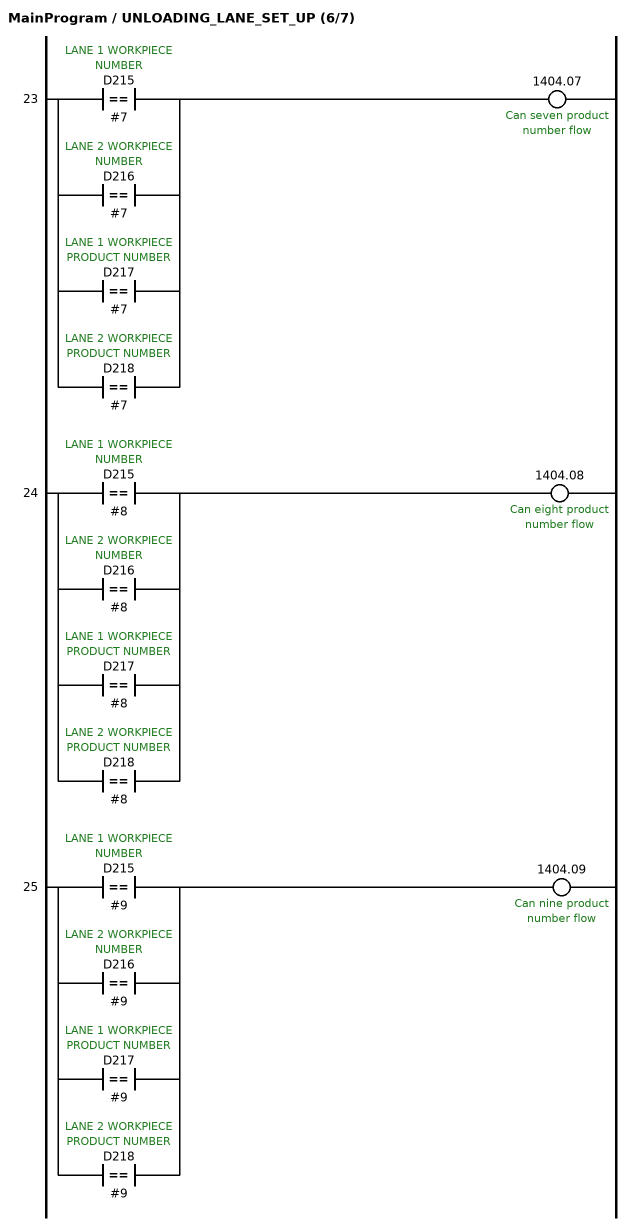
; [picture p192: MainProgram / UNLOADING_LANE_SET_UP, rungs 23-25]
; rung 23
LD=(300) D215 #7  ; LANE 1 WORKPIECE NUMBER
OR=(300) D216 #7  ; LANE 2 WORKPIECE NUMBER
OR=(300) D217 #7  ; LANE 1 WORKPIECE PRODUCT NUMBER
OR=(300) D218 #7  ; LANE 2 WORKPIECE PRODUCT NUMBER
OUT 1404.07  ; Can seven product number flow
; rung 24
LD=(300) D215 #8  ; LANE 1 WORKPIECE NUMBER
OR=(300) D216 #8  ; LANE 2 WORKPIECE NUMBER
OR=(300) D217 #8  ; LANE 1 WORKPIECE PRODUCT NUMBER
OR=(300) D218 #8  ; LANE 2 WORKPIECE PRODUCT NUMBER
OUT 1404.08  ; Can eight product number flow
; rung 25
LD=(300) D215 #9  ; LANE 1 WORKPIECE NUMBER
OR=(300) D216 #9  ; LANE 2 WORKPIECE NUMBER
OR=(300) D217 #9  ; LANE 1 WORKPIECE PRODUCT NUMBER
OR=(300) D218 #9  ; LANE 2 WORKPIECE PRODUCT NUMBER
OUT 1404.09  ; Can nine product number flow

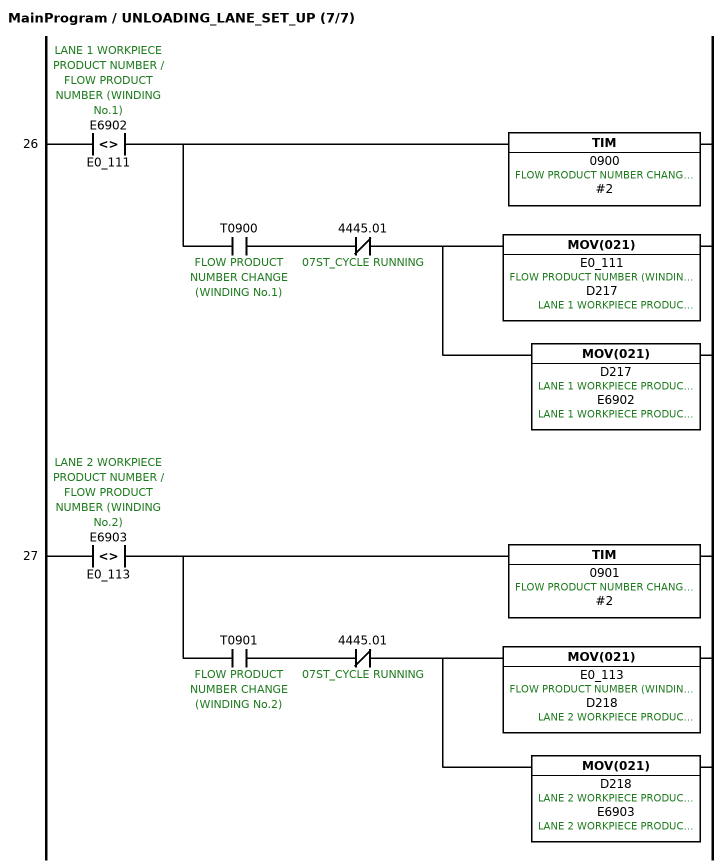
; rung 26
LD<>(305) E6902 E0_111  ; LANE 1 WORKPIECE PRODUCT NUMBER, FLOW PRODUCT NUMBER (WINDING No.1)
TIM 0900 #2  ; FLOW PRODUCT NUMBER CHANGE (WINDING No.1)
AND T0900  ; FLOW PRODUCT NUMBER CHANGE (WINDING No.1)
ANDNOT 4445.01  ; 07ST_CYCLE RUNNING
MOV(021) E0_111 D217  ; FLOW PRODUCT NUMBER (WINDING No.1), LANE 1 WORKPIECE PRODUCT NUMBER
MOV(021) D217 E6902  ; LANE 1 WORKPIECE PRODUCT NUMBER
; rung 27
LD<>(305) E6903 E0_113  ; LANE 2 WORKPIECE PRODUCT NUMBER, FLOW PRODUCT NUMBER (WINDING No.2)
TIM 0901 #2  ; FLOW PRODUCT NUMBER CHANGE (WINDING No.2)
AND T0901  ; FLOW PRODUCT NUMBER CHANGE (WINDING No.2)
ANDNOT 4445.01  ; 07ST_CYCLE RUNNING
MOV(021) E0_113 D218  ; FLOW PRODUCT NUMBER (WINDING No.2), LANE 2 WORKPIECE PRODUCT NUMBER
MOV(021) D218 E6903  ; LANE 2 WORKPIECE PRODUCT NUMBER

### Section WORKPIECE_NUMBER_SET_UP

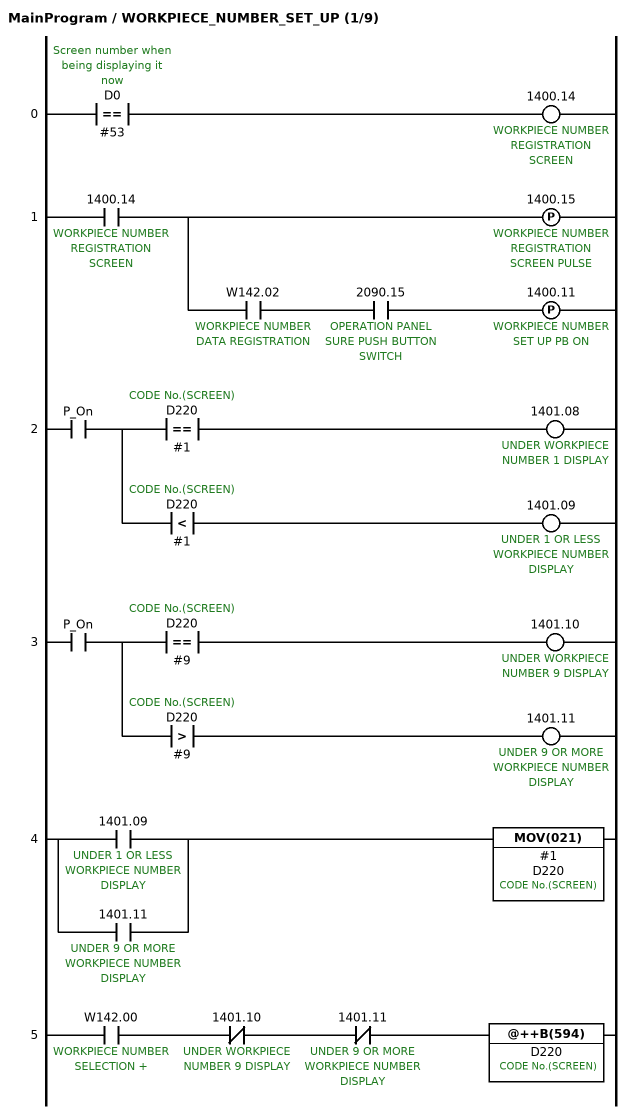
; rung 0
LD=(300) D0 #53  ; Screen number when being displaying it now
OUT 1400.14  ; WORKPIECE NUMBER REGISTRATION SCREEN
; rung 1
LD 1400.14  ; WORKPIECE NUMBER REGISTRATION SCREEN
DIFU(013) 1400.15  ; WORKPIECE NUMBER REGISTRATION SCREEN PULSE
AND W142.02  ; WORKPIECE NUMBER DATA REGISTRATION
AND 2090.15  ; OPERATION PANEL SURE PUSH BUTTON SWITCH
DIFU(013) 1400.11  ; WORKPIECE NUMBER SET UP PB ON
; rung 2
LD P_On
OUT TR0
AND=(300) D220 #1  ; CODE No.(SCREEN)
OUT 1401.08  ; UNDER WORKPIECE NUMBER 1 DISPLAY
LD TR0
AND<(310) D220 #1  ; CODE No.(SCREEN)
OUT 1401.09  ; UNDER 1 OR LESS WORKPIECE NUMBER DISPLAY
; rung 3
LD P_On
OUT TR0
AND=(300) D220 #9  ; CODE No.(SCREEN)
OUT 1401.10  ; UNDER WORKPIECE NUMBER 9 DISPLAY
LD TR0
AND>(320) D220 #9  ; CODE No.(SCREEN)
OUT 1401.11  ; UNDER 9 OR MORE WORKPIECE NUMBER DISPLAY
; rung 4
LD 1401.09  ; UNDER 1 OR LESS WORKPIECE NUMBER DISPLAY
OR 1401.11  ; UNDER 9 OR MORE WORKPIECE NUMBER DISPLAY
MOV(021) #1 D220  ; CODE No.(SCREEN)
; rung 5
LD W142.00  ; WORKPIECE NUMBER SELECTION +
ANDNOT 1401.10  ; UNDER WORKPIECE NUMBER 9 DISPLAY
ANDNOT 1401.11  ; UNDER 9 OR MORE WORKPIECE NUMBER DISPLAY
@++B(594) D220  ; CODE No.(SCREEN)

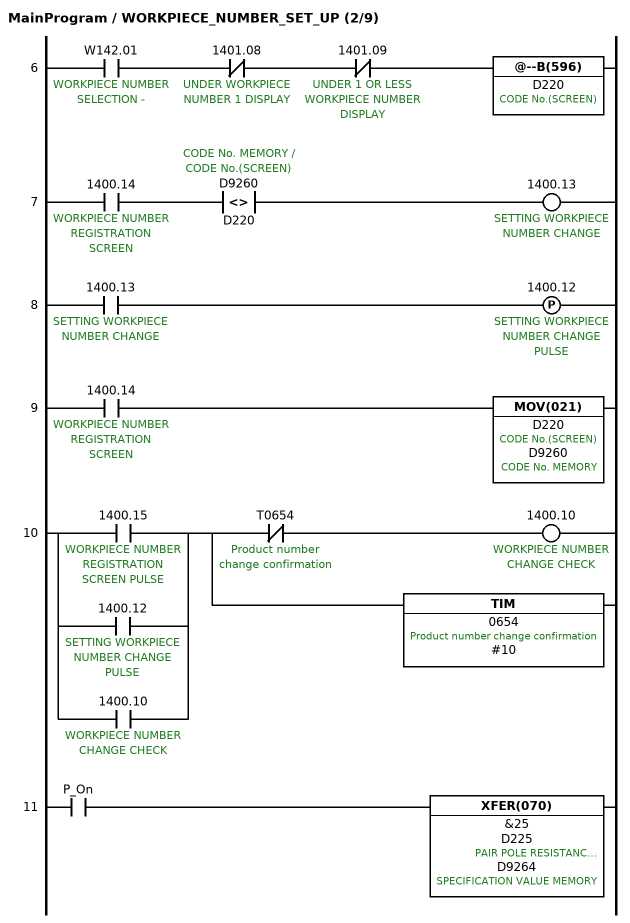
; rung 6
LD W142.01  ; WORKPIECE NUMBER SELECTION -
ANDNOT 1401.08  ; UNDER WORKPIECE NUMBER 1 DISPLAY
ANDNOT 1401.09  ; UNDER 1 OR LESS WORKPIECE NUMBER DISPLAY
@--B(596) D220  ; CODE No.(SCREEN)
; rung 7
LD 1400.14  ; WORKPIECE NUMBER REGISTRATION SCREEN
AND<>(305) D9260 D220  ; CODE No. MEMORY, CODE No.(SCREEN)
OUT 1400.13  ; SETTING WORKPIECE NUMBER CHANGE
; rung 8
LD 1400.13  ; SETTING WORKPIECE NUMBER CHANGE
DIFU(013) 1400.12  ; SETTING WORKPIECE NUMBER CHANGE PULSE
; rung 9
LD 1400.14  ; WORKPIECE NUMBER REGISTRATION SCREEN
MOV(021) D220 D9260  ; CODE No.(SCREEN), CODE No. MEMORY
; rung 10
LD 1400.15  ; WORKPIECE NUMBER REGISTRATION SCREEN PULSE
OR 1400.12  ; SETTING WORKPIECE NUMBER CHANGE PULSE
OR 1400.10  ; WORKPIECE NUMBER CHANGE CHECK
OUT TR0
ANDNOT T0654  ; Product number change confirmation
OUT 1400.10  ; WORKPIECE NUMBER CHANGE CHECK
LD TR0
TIM 0654 #10  ; Product number change confirmation
; rung 11
LD P_On
XFER(070) &25 D225 D9264  ; PAIR POLE RESISTANCE SPECIFICATION MINIMUM VALUE(SCREEN), SPECIFICATION VALUE MEMORY

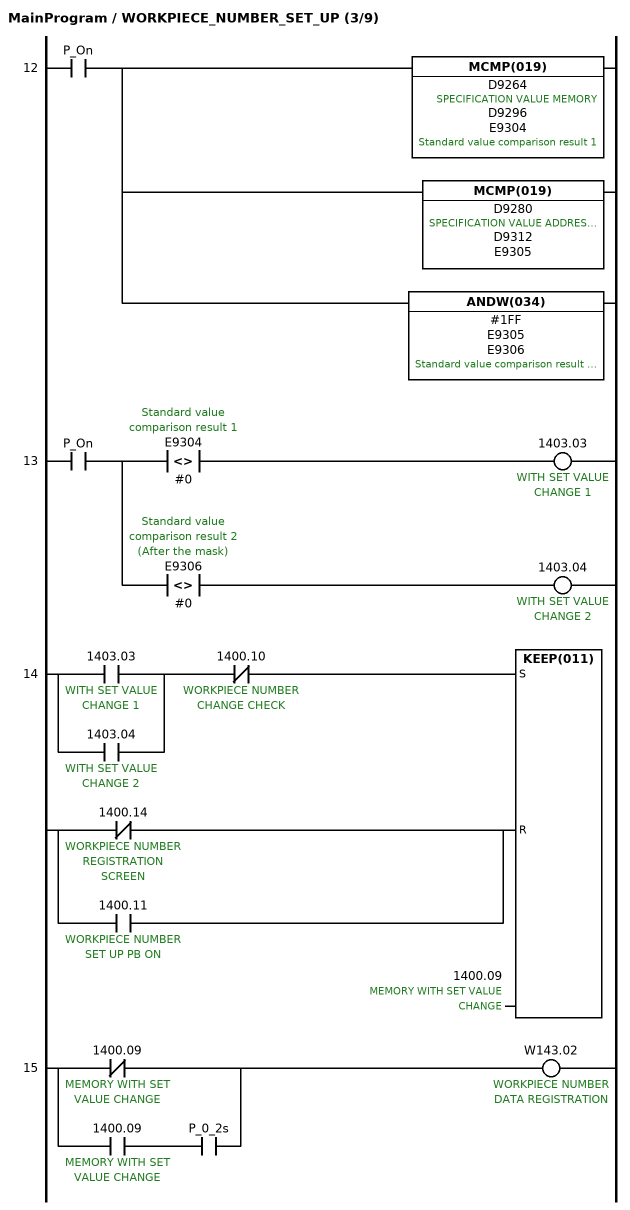
; rung 12
LD P_On
MCMP(019) D9264 D9296 E9304  ; SPECIFICATION VALUE MEMORY, Standard value comparison result 1
MCMP(019) D9280 D9312 E9305  ; SPECIFICATION VALUE ADDRESS INDIRECT SPECIFICATION
ANDW(034) #1FF E9305 E9306  ; Standard value comparison result 2 (After the mask)
; rung 13
LD P_On
OUT TR0
AND<>(305) E9304 #0  ; Standard value comparison result 1
OUT 1403.03  ; WITH SET VALUE CHANGE 1
LD TR0
AND<>(305) E9306 #0  ; Standard value comparison result 2 (After the mask)
OUT 1403.04  ; WITH SET VALUE CHANGE 2
; rung 14
LD 1403.03  ; WITH SET VALUE CHANGE 1
OR 1403.04  ; WITH SET VALUE CHANGE 2
ANDNOT 1400.10  ; WORKPIECE NUMBER CHANGE CHECK
LDNOT 1400.14  ; WORKPIECE NUMBER REGISTRATION SCREEN
OR 1400.11  ; WORKPIECE NUMBER SET UP PB ON
KEEP(011) 1400.09  ; MEMORY WITH SET VALUE CHANGE
; rung 15
LDNOT 1400.09  ; MEMORY WITH SET VALUE CHANGE
LD 1400.09  ; MEMORY WITH SET VALUE CHANGE
AND P_0_2s
ORLD
OUT W143.02  ; WORKPIECE NUMBER DATA REGISTRATION

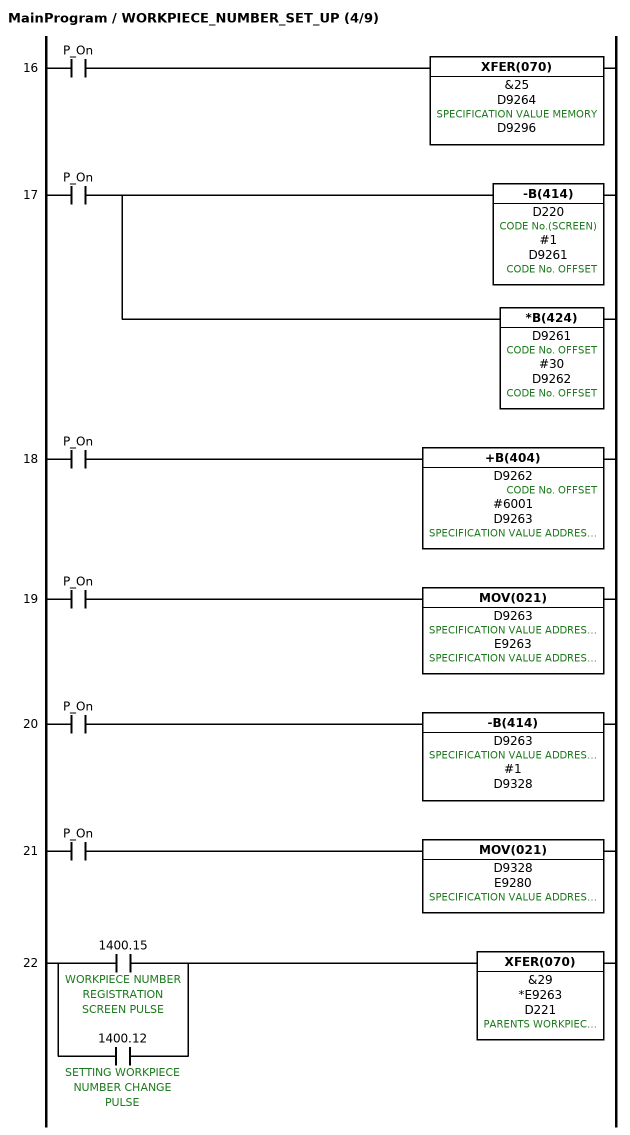
; rung 16
LD P_On
XFER(070) &25 D9264 D9296  ; SPECIFICATION VALUE MEMORY
; rung 17
LD P_On
-B(414) D220 #1 D9261  ; CODE No.(SCREEN), CODE No. OFFSET
*B(424) D9261 #30 D9262  ; CODE No. OFFSET
; rung 18
LD P_On
+B(404) D9262 #6001 D9263  ; CODE No. OFFSET, SPECIFICATION VALUE ADDRESS INDIRECT SPECIFICATION
; rung 19
LD P_On
MOV(021) D9263 E9263  ; SPECIFICATION VALUE ADDRESS INDIRECT SPECIFICATION
; rung 20
LD P_On
-B(414) D9263 #1 D9328  ; SPECIFICATION VALUE ADDRESS INDIRECT SPECIFICATION
; rung 21
LD P_On
MOV(021) D9328 E9280  ; SPECIFICATION VALUE ADDRESS INDIRECT SPECIFICATION
; rung 22
LD 1400.15  ; WORKPIECE NUMBER REGISTRATION SCREEN PULSE
OR 1400.12  ; SETTING WORKPIECE NUMBER CHANGE PULSE
XFER(070) &29 *E9263 D221  ; PARENTS WORKPIECE NUMBER(SCREEN)

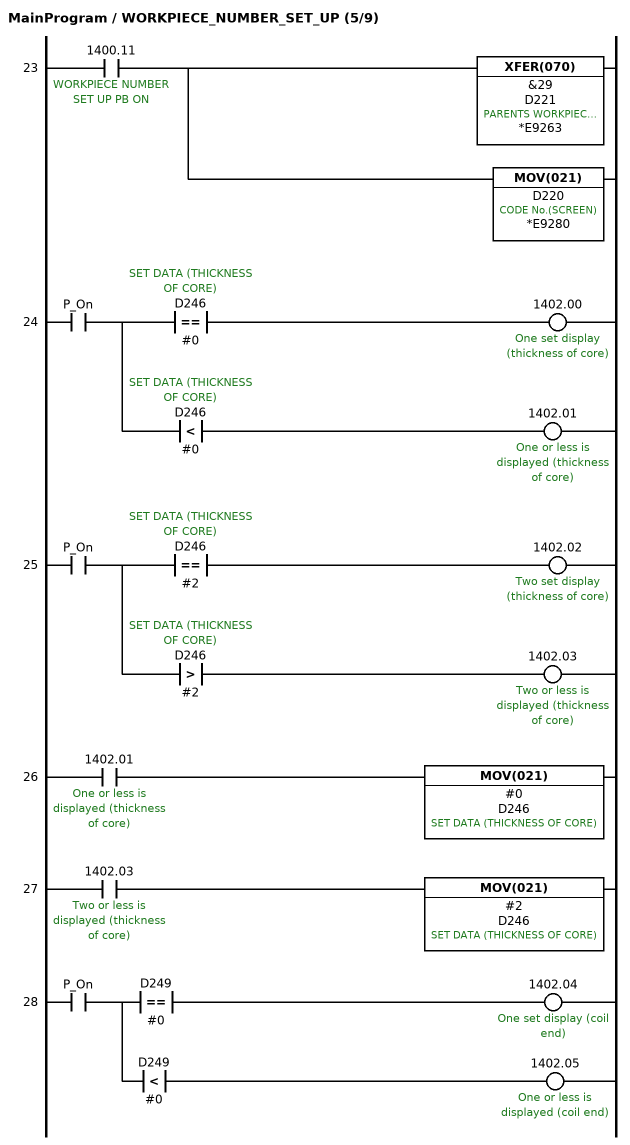
; rung 23
LD 1400.11  ; WORKPIECE NUMBER SET UP PB ON
XFER(070) &29 D221 *E9263  ; PARENTS WORKPIECE NUMBER(SCREEN)
MOV(021) D220 *E9280  ; CODE No.(SCREEN)
; rung 24
LD P_On
OUT TR0
AND=(300) D246 #0  ; SET DATA (THICKNESS OF CORE)
OUT 1402.00  ; One set display (thickness of core)
LD TR0
AND<(310) D246 #0  ; SET DATA (THICKNESS OF CORE)
OUT 1402.01  ; One or less is displayed (thickness of core)
; rung 25
LD P_On
OUT TR0
AND=(300) D246 #2  ; SET DATA (THICKNESS OF CORE)
OUT 1402.02  ; Two set display (thickness of core)
LD TR0
AND>(320) D246 #2  ; SET DATA (THICKNESS OF CORE)
OUT 1402.03  ; Two or less is displayed (thickness of core)
; rung 26
LD 1402.01  ; One or less is displayed (thickness of core)
MOV(021) #0 D246  ; SET DATA (THICKNESS OF CORE)
; rung 27
LD 1402.03  ; Two or less is displayed (thickness of core)
MOV(021) #2 D246  ; SET DATA (THICKNESS OF CORE)
; rung 28
LD P_On
OUT TR0
AND=(300) D249 #0
OUT 1402.04  ; One set display (coil end)
LD TR0
AND<(310) D249 #0
OUT 1402.05  ; One or less is displayed (coil end)

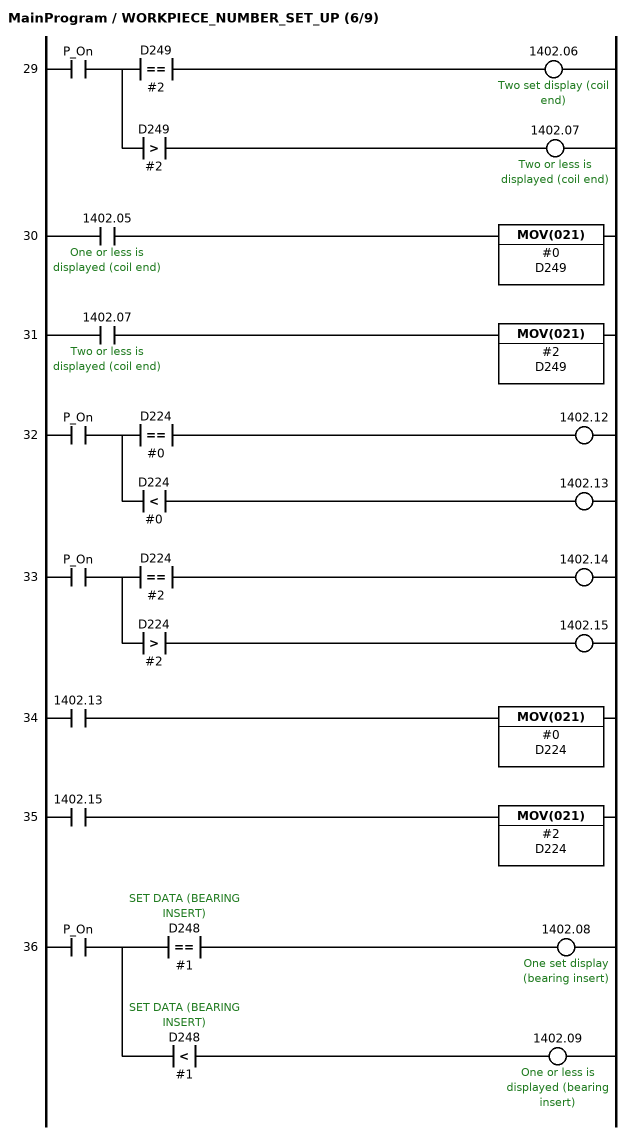
; rung 29
LD P_On
OUT TR0
AND=(300) D249 #2
OUT 1402.06  ; Two set display (coil end)
LD TR0
AND>(320) D249 #2
OUT 1402.07  ; Two or less is displayed (coil end)
; rung 30
LD 1402.05  ; One or less is displayed (coil end)
MOV(021) #0 D249
; rung 31
LD 1402.07  ; Two or less is displayed (coil end)
MOV(021) #2 D249
; rung 32
LD P_On
OUT TR0
AND=(300) D224 #0
OUT 1402.12
LD TR0
AND<(310) D224 #0
OUT 1402.13
; rung 33
LD P_On
OUT TR0
AND=(300) D224 #2
OUT 1402.14
LD TR0
AND>(320) D224 #2
OUT 1402.15
; rung 34
LD 1402.13
MOV(021) #0 D224
; rung 35
LD 1402.15
MOV(021) #2 D224
; rung 36
LD P_On
OUT TR0
AND=(300) D248 #1  ; SET DATA (BEARING INSERT)
OUT 1402.08  ; One set display (bearing insert)
LD TR0
AND<(310) D248 #1  ; SET DATA (BEARING INSERT)
OUT 1402.09  ; One or less is displayed (bearing insert)

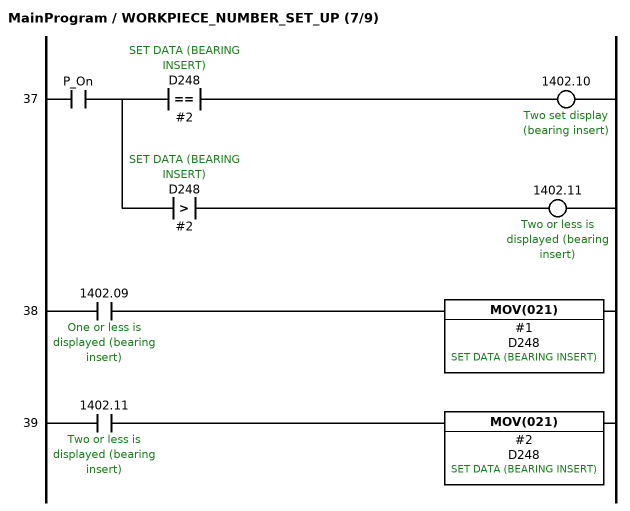
; rung 37
LD P_On
OUT TR0
AND=(300) D248 #2  ; SET DATA (BEARING INSERT)
OUT 1402.10  ; Two set display (bearing insert)
LD TR0
AND>(320) D248 #2  ; SET DATA (BEARING INSERT)
OUT 1402.11  ; Two or less is displayed (bearing insert)
; rung 38
LD 1402.09  ; One or less is displayed (bearing insert)
MOV(021) #1 D248  ; SET DATA (BEARING INSERT)
; rung 39
LD 1402.11  ; Two or less is displayed (bearing insert)
MOV(021) #2 D248  ; SET DATA (BEARING INSERT)

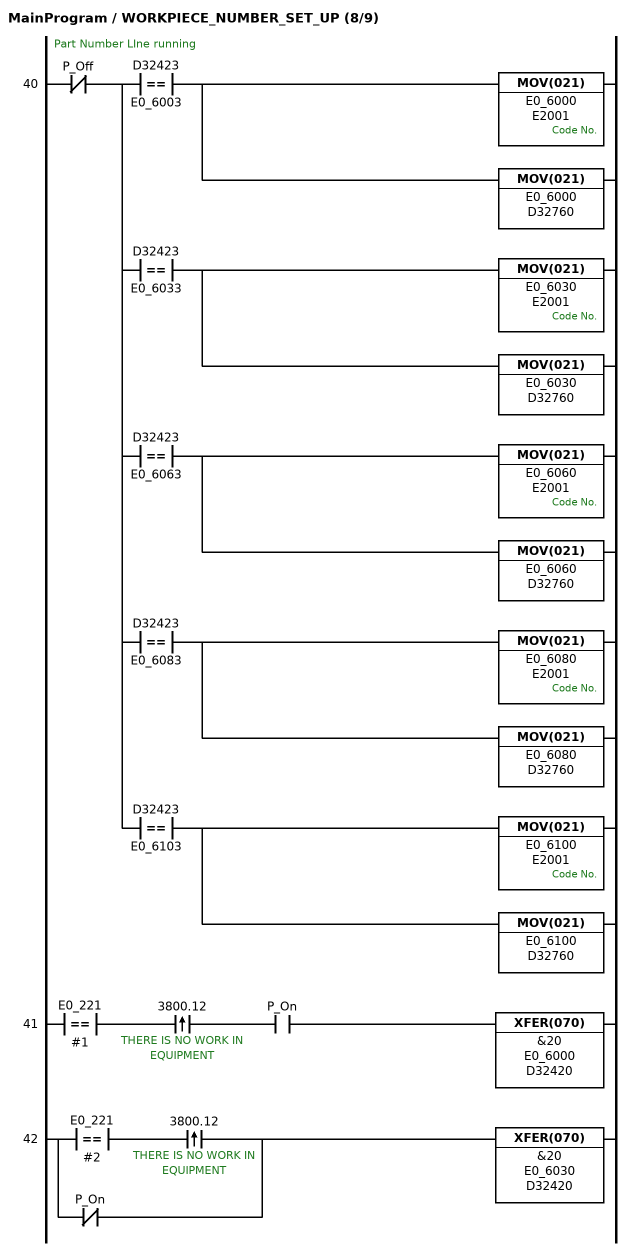
; rung 40: Part Number LIne running
LDNOT P_Off
OUT TR0
AND=(300) D32423 E0_6003
MOV(021) E0_6000 E2001  ; Code No.
MOV(021) E0_6000 D32760
LD TR0
AND=(300) D32423 E0_6033
MOV(021) E0_6030 E2001  ; Code No.
MOV(021) E0_6030 D32760
LD TR0
AND=(300) D32423 E0_6063
MOV(021) E0_6060 E2001  ; Code No.
MOV(021) E0_6060 D32760
LD TR0
AND=(300) D32423 E0_6083
MOV(021) E0_6080 E2001  ; Code No.
MOV(021) E0_6080 D32760
LD TR0
AND=(300) D32423 E0_6103
MOV(021) E0_6100 E2001  ; Code No.
MOV(021) E0_6100 D32760
; rung 41
LD=(300) E0_221 #1
@AND 3800.12  ; THERE IS NO WORK IN EQUIPMENT
AND P_On
XFER(070) &20 E0_6000 D32420
; rung 42
LD=(300) E0_221 #2
@AND 3800.12  ; THERE IS NO WORK IN EQUIPMENT
ORNOT P_On
XFER(070) &20 E0_6030 D32420

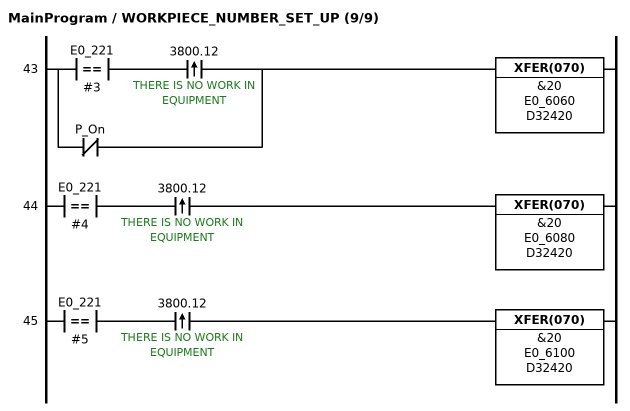
; rung 43
LD=(300) E0_221 #3
@AND 3800.12  ; THERE IS NO WORK IN EQUIPMENT
ORNOT P_On
XFER(070) &20 E0_6060 D32420
; rung 44
LD=(300) E0_221 #4
@AND 3800.12  ; THERE IS NO WORK IN EQUIPMENT
XFER(070) &20 E0_6080 D32420
; rung 45
LD=(300) E0_221 #5
@AND 3800.12  ; THERE IS NO WORK IN EQUIPMENT
XFER(070) &20 E0_6100 D32420

### Section RC5_CONTROLLER_STARTING

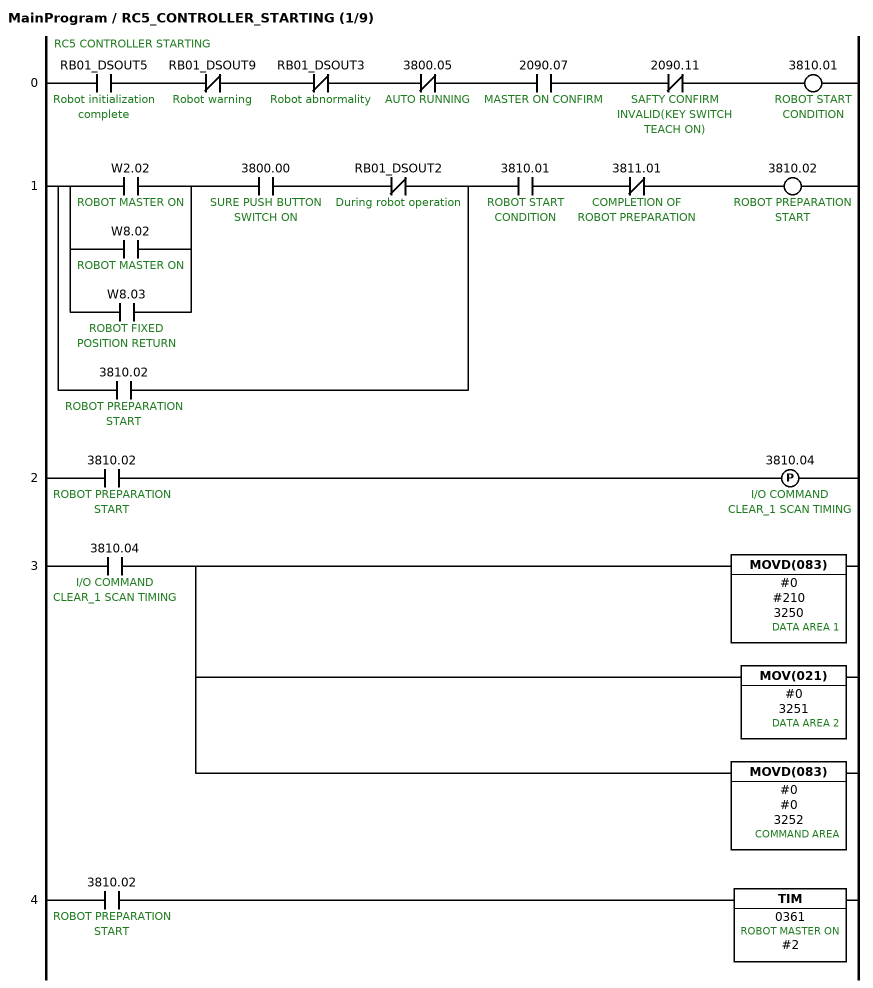
; rung 0: RC5 CONTROLLER STARTING
LD RB01_DSOUT5  ; Robot initialization complete
ANDNOT RB01_DSOUT9  ; Robot warning
ANDNOT RB01_DSOUT3  ; Robot abnormality
ANDNOT 3800.05  ; AUTO RUNNING
AND 2090.07  ; MASTER ON CONFIRM
ANDNOT 2090.11  ; SAFTY CONFIRM INVALID(KEY SWITCH TEACH ON)
OUT 3810.01  ; ROBOT START CONDITION
; rung 1
LD W2.02  ; ROBOT MASTER ON
OR W8.02  ; ROBOT MASTER ON
OR W8.03  ; ROBOT FIXED POSITION RETURN
AND 3800.00  ; SURE PUSH BUTTON SWITCH ON
ANDNOT RB01_DSOUT2  ; During robot operation
OR 3810.02  ; ROBOT PREPARATION START
AND 3810.01  ; ROBOT START CONDITION
ANDNOT 3811.01  ; COMPLETION OF ROBOT PREPARATION
OUT 3810.02  ; ROBOT PREPARATION START
; rung 2
LD 3810.02  ; ROBOT PREPARATION START
DIFU(013) 3810.04  ; I/O COMMAND CLEAR_1 SCAN TIMING
; rung 3
LD 3810.04  ; I/O COMMAND CLEAR_1 SCAN TIMING
MOVD(083) #0 #210 3250  ; DATA AREA 1
MOV(021) #0 3251  ; DATA AREA 2
MOVD(083) #0 #0 3252  ; COMMAND AREA
; rung 4
LD 3810.02  ; ROBOT PREPARATION START
TIM 0361 #2  ; ROBOT MASTER ON

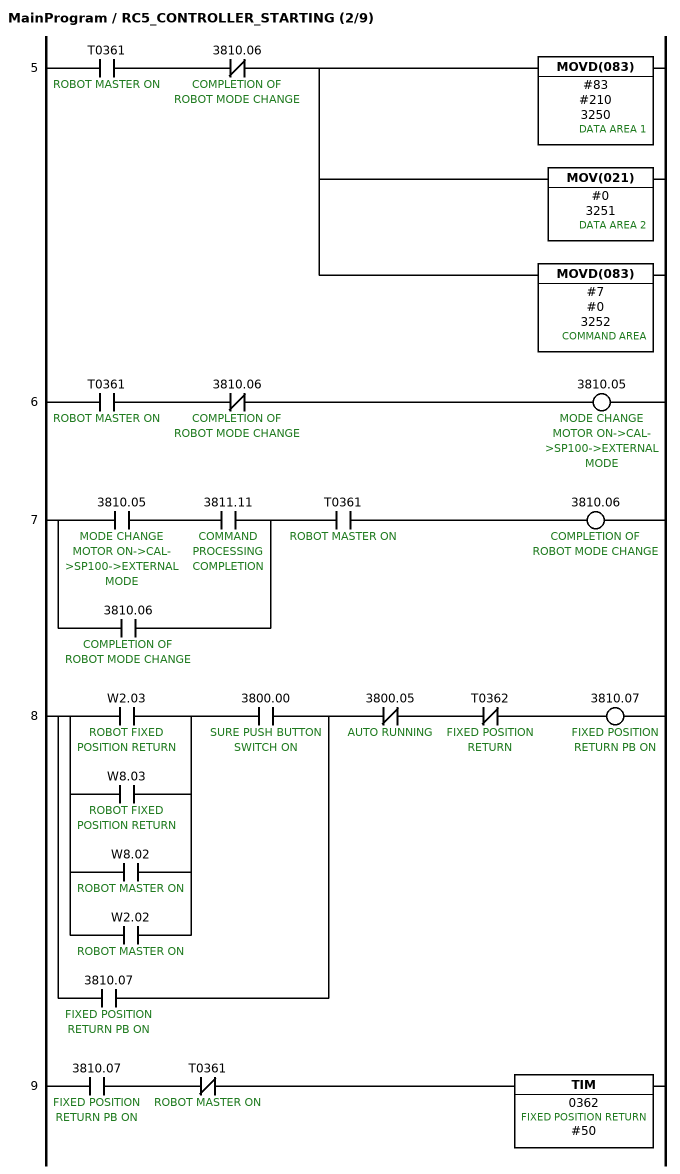
; rung 5
LD T0361  ; ROBOT MASTER ON
ANDNOT 3810.06  ; COMPLETION OF ROBOT MODE CHANGE
MOVD(083) #83 #210 3250  ; DATA AREA 1
MOV(021) #0 3251  ; DATA AREA 2
MOVD(083) #7 #0 3252  ; COMMAND AREA
; rung 6
LD T0361  ; ROBOT MASTER ON
ANDNOT 3810.06  ; COMPLETION OF ROBOT MODE CHANGE
OUT 3810.05  ; MODE CHANGE MOTOR ON->CAL->SP100->EXTERNAL MODE
; rung 7
LD 3810.05  ; MODE CHANGE MOTOR ON->CAL->SP100->EXTERNAL MODE
AND 3811.11  ; COMMAND PROCESSING COMPLETION
OR 3810.06  ; COMPLETION OF ROBOT MODE CHANGE
AND T0361  ; ROBOT MASTER ON
OUT 3810.06  ; COMPLETION OF ROBOT MODE CHANGE
; rung 8
LD W2.03  ; ROBOT FIXED POSITION RETURN
OR W8.03  ; ROBOT FIXED POSITION RETURN
OR W8.02  ; ROBOT MASTER ON
OR W2.02  ; ROBOT MASTER ON
AND 3800.00  ; SURE PUSH BUTTON SWITCH ON
OR 3810.07  ; FIXED POSITION RETURN PB ON
ANDNOT 3800.05  ; AUTO RUNNING
ANDNOT T0362  ; FIXED POSITION RETURN
OUT 3810.07  ; FIXED POSITION RETURN PB ON
; rung 9
LD 3810.07  ; FIXED POSITION RETURN PB ON
ANDNOT T0361  ; ROBOT MASTER ON
TIM 0362 #50  ; FIXED POSITION RETURN

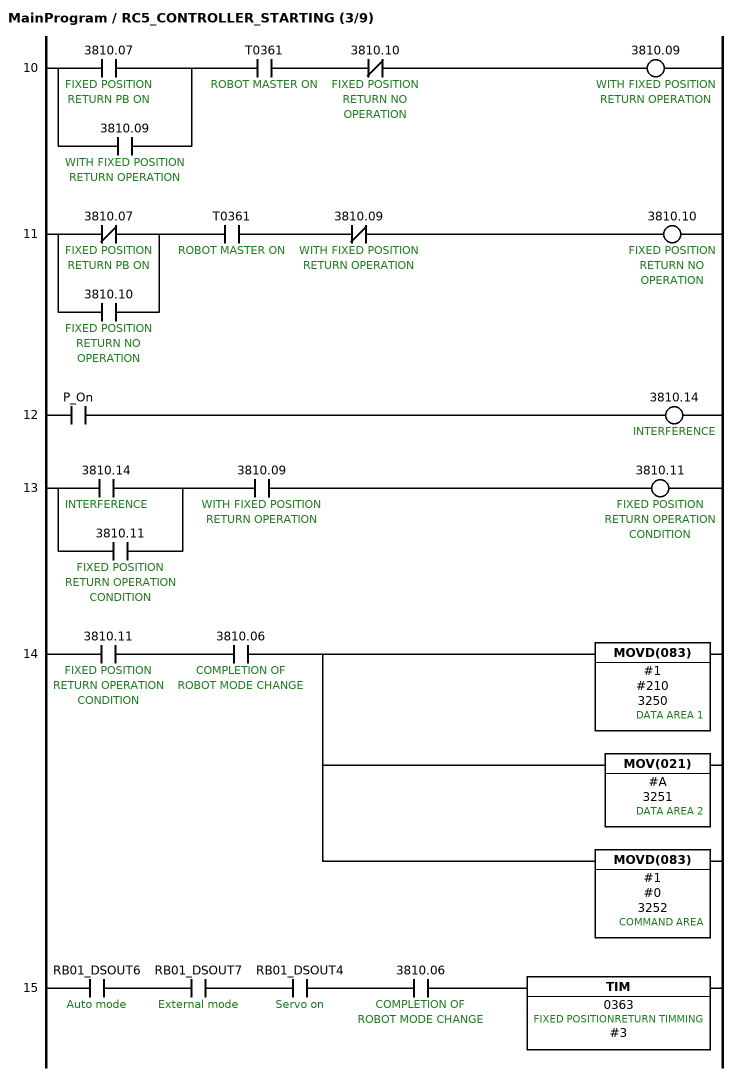
; rung 10
LD 3810.07  ; FIXED POSITION RETURN PB ON
OR 3810.09  ; WITH FIXED POSITION RETURN OPERATION
AND T0361  ; ROBOT MASTER ON
ANDNOT 3810.10  ; FIXED POSITION RETURN NO OPERATION
OUT 3810.09  ; WITH FIXED POSITION RETURN OPERATION
; rung 11
LDNOT 3810.07  ; FIXED POSITION RETURN PB ON
OR 3810.10  ; FIXED POSITION RETURN NO OPERATION
AND T0361  ; ROBOT MASTER ON
ANDNOT 3810.09  ; WITH FIXED POSITION RETURN OPERATION
OUT 3810.10  ; FIXED POSITION RETURN NO OPERATION
; rung 12
LD P_On
OUT 3810.14  ; INTERFERENCE
; rung 13
LD 3810.14  ; INTERFERENCE
OR 3810.11  ; FIXED POSITION RETURN OPERATION CONDITION
AND 3810.09  ; WITH FIXED POSITION RETURN OPERATION
OUT 3810.11  ; FIXED POSITION RETURN OPERATION CONDITION
; rung 14
LD 3810.11  ; FIXED POSITION RETURN OPERATION CONDITION
AND 3810.06  ; COMPLETION OF ROBOT MODE CHANGE
MOVD(083) #1 #210 3250  ; DATA AREA 1
MOV(021) #A 3251  ; DATA AREA 2
MOVD(083) #1 #0 3252  ; COMMAND AREA
; rung 15
LD RB01_DSOUT6  ; Auto mode
AND RB01_DSOUT7  ; External mode
AND RB01_DSOUT4  ; Servo on
AND 3810.06  ; COMPLETION OF ROBOT MODE CHANGE
TIM 0363 #3  ; FIXED POSITIONRETURN TIMMING

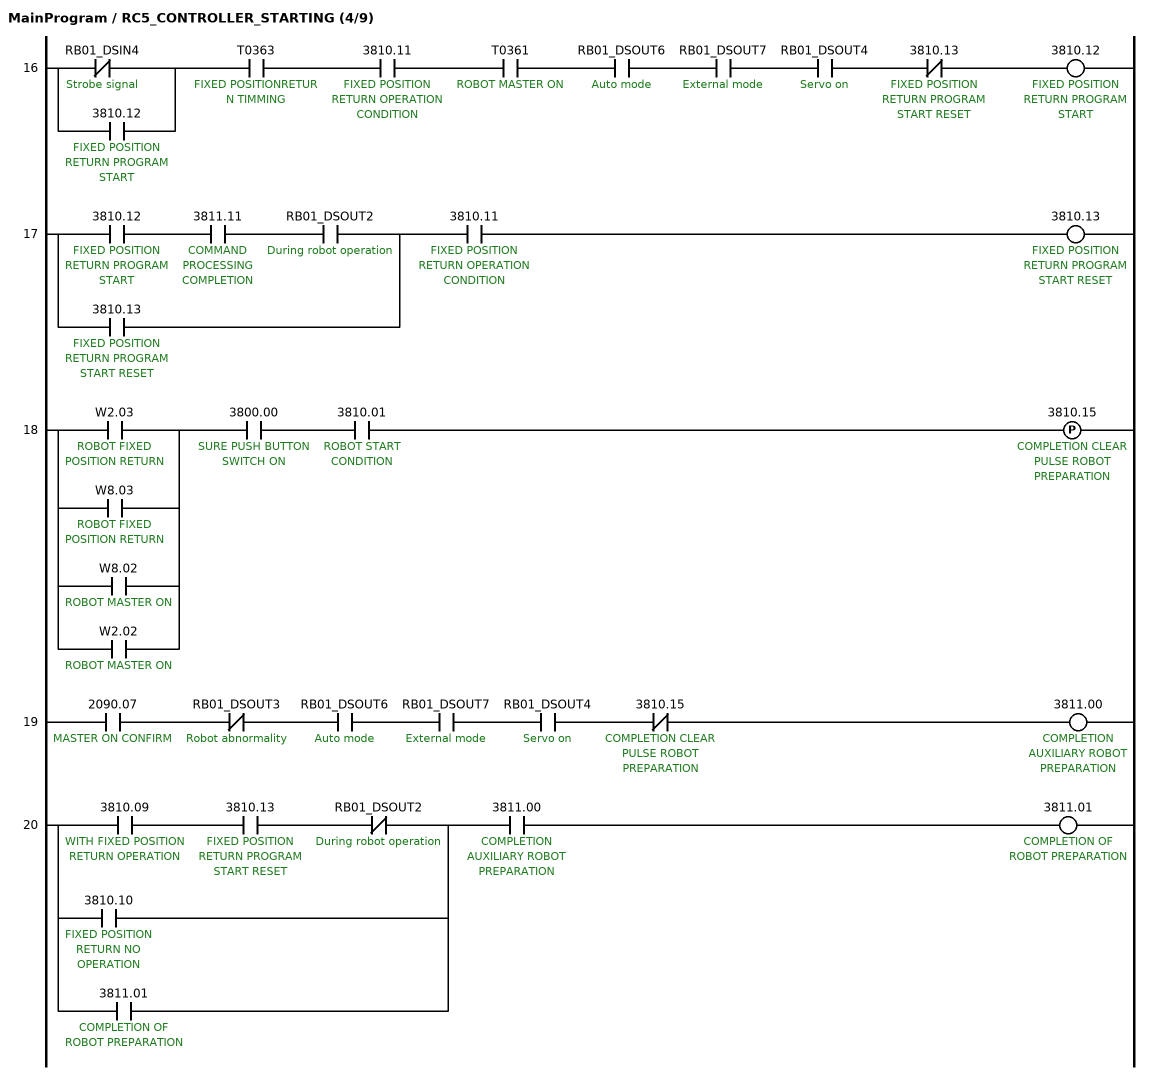
; rung 16
LDNOT RB01_DSIN4  ; Strobe signal
OR 3810.12  ; FIXED POSITION RETURN PROGRAM START
AND T0363  ; FIXED POSITIONRETURN TIMMING
AND 3810.11  ; FIXED POSITION RETURN OPERATION CONDITION
AND T0361  ; ROBOT MASTER ON
AND RB01_DSOUT6  ; Auto mode
AND RB01_DSOUT7  ; External mode
AND RB01_DSOUT4  ; Servo on
ANDNOT 3810.13  ; FIXED POSITION RETURN PROGRAM START RESET
OUT 3810.12  ; FIXED POSITION RETURN PROGRAM START
; rung 17
LD 3810.12  ; FIXED POSITION RETURN PROGRAM START
AND 3811.11  ; COMMAND PROCESSING COMPLETION
AND RB01_DSOUT2  ; During robot operation
OR 3810.13  ; FIXED POSITION RETURN PROGRAM START RESET
AND 3810.11  ; FIXED POSITION RETURN OPERATION CONDITION
OUT 3810.13  ; FIXED POSITION RETURN PROGRAM START RESET
; rung 18
LD W2.03  ; ROBOT FIXED POSITION RETURN
OR W8.03  ; ROBOT FIXED POSITION RETURN
OR W8.02  ; ROBOT MASTER ON
OR W2.02  ; ROBOT MASTER ON
AND 3800.00  ; SURE PUSH BUTTON SWITCH ON
AND 3810.01  ; ROBOT START CONDITION
DIFU(013) 3810.15  ; COMPLETION CLEAR PULSE ROBOT PREPARATION
; rung 19
LD 2090.07  ; MASTER ON CONFIRM
ANDNOT RB01_DSOUT3  ; Robot abnormality
AND RB01_DSOUT6  ; Auto mode
AND RB01_DSOUT7  ; External mode
AND RB01_DSOUT4  ; Servo on
ANDNOT 3810.15  ; COMPLETION CLEAR PULSE ROBOT PREPARATION
OUT 3811.00  ; COMPLETION AUXILIARY ROBOT PREPARATION
; rung 20
LD 3810.09  ; WITH FIXED POSITION RETURN OPERATION
AND 3810.13  ; FIXED POSITION RETURN PROGRAM START RESET
ANDNOT RB01_DSOUT2  ; During robot operation
OR 3810.10  ; FIXED POSITION RETURN NO OPERATION
OR 3811.01  ; COMPLETION OF ROBOT PREPARATION
AND 3811.00  ; COMPLETION AUXILIARY ROBOT PREPARATION
OUT 3811.01  ; COMPLETION OF ROBOT PREPARATION

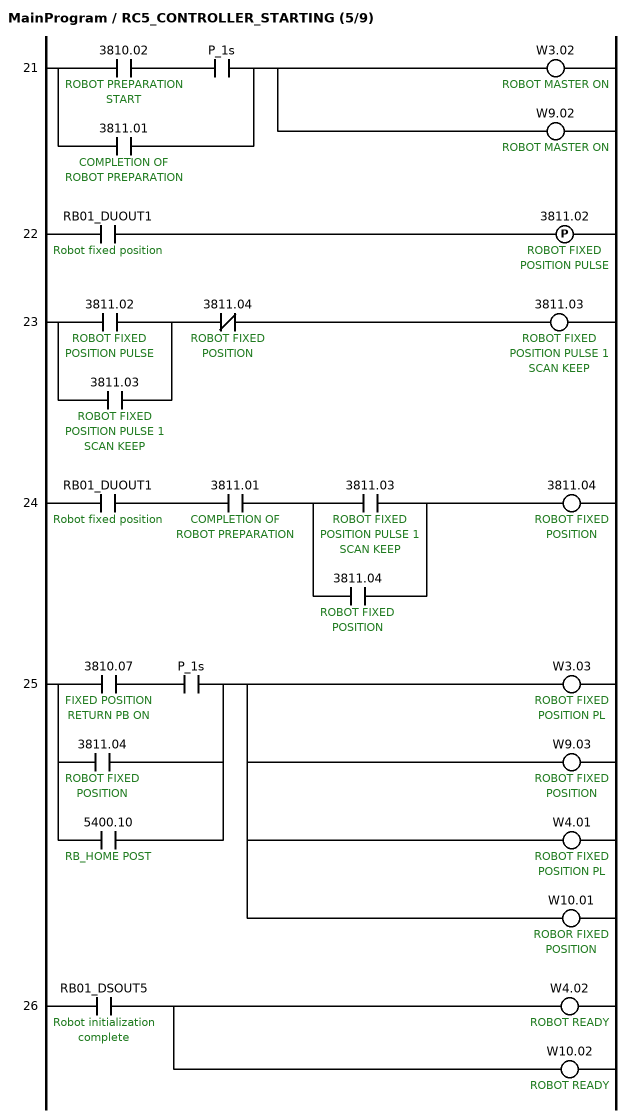
; rung 21
LD 3810.02  ; ROBOT PREPARATION START
AND P_1s
OR 3811.01  ; COMPLETION OF ROBOT PREPARATION
OUT W3.02  ; ROBOT MASTER ON
OUT W9.02  ; ROBOT MASTER ON
; rung 22
LD RB01_DUOUT1  ; Robot fixed position
DIFU(013) 3811.02  ; ROBOT FIXED POSITION PULSE
; rung 23
LD 3811.02  ; ROBOT FIXED POSITION PULSE
OR 3811.03  ; ROBOT FIXED POSITION PULSE 1 SCAN KEEP
ANDNOT 3811.04  ; ROBOT FIXED POSITION
OUT 3811.03  ; ROBOT FIXED POSITION PULSE 1 SCAN KEEP
; rung 24
LD RB01_DUOUT1  ; Robot fixed position
AND 3811.01  ; COMPLETION OF ROBOT PREPARATION
LD 3811.03  ; ROBOT FIXED POSITION PULSE 1 SCAN KEEP
OR 3811.04  ; ROBOT FIXED POSITION
ANDLD
OUT 3811.04  ; ROBOT FIXED POSITION
; rung 25
LD 3810.07  ; FIXED POSITION RETURN PB ON
AND P_1s
OR 3811.04  ; ROBOT FIXED POSITION
OR 5400.10  ; RB_HOME POST
OUT W3.03  ; ROBOT FIXED POSITION PL
OUT W9.03  ; ROBOT FIXED POSITION
OUT W4.01  ; ROBOT FIXED POSITION PL
OUT W10.01  ; ROBOR FIXED POSITION
; rung 26
LD RB01_DSOUT5  ; Robot initialization complete
OUT W4.02  ; ROBOT READY
OUT W10.02  ; ROBOT READY

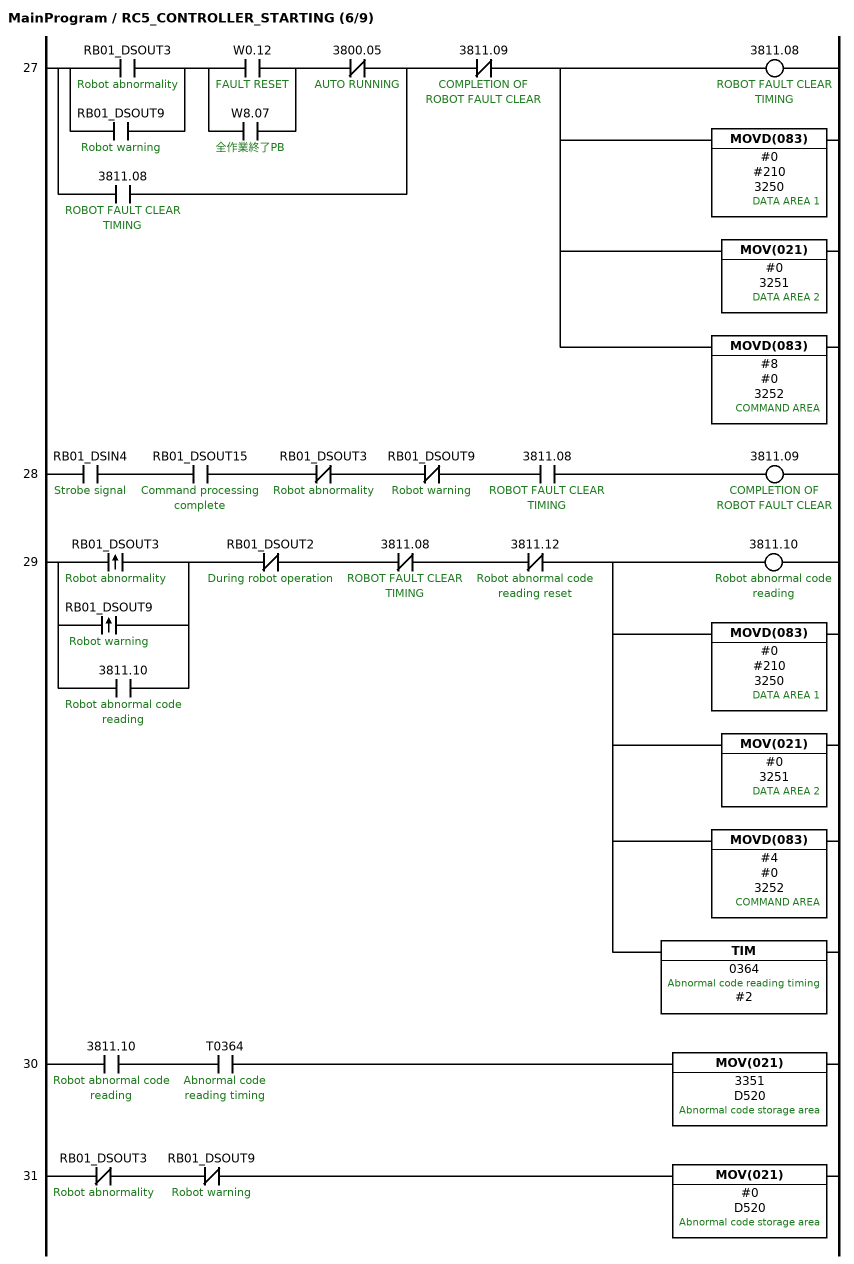
; rung 27
LD RB01_DSOUT3  ; Robot abnormality
OR RB01_DSOUT9  ; Robot warning
LD W0.12  ; FAULT RESET
OR W8.07  ; 全作業終了PB
ANDLD
ANDNOT 3800.05  ; AUTO RUNNING
OR 3811.08  ; ROBOT FAULT CLEAR TIMING
ANDNOT 3811.09  ; COMPLETION OF ROBOT FAULT CLEAR
OUT 3811.08  ; ROBOT FAULT CLEAR TIMING
MOVD(083) #0 #210 3250  ; DATA AREA 1
MOV(021) #0 3251  ; DATA AREA 2
MOVD(083) #8 #0 3252  ; COMMAND AREA
; rung 28
LD RB01_DSIN4  ; Strobe signal
AND RB01_DSOUT15  ; Command processing complete
ANDNOT RB01_DSOUT3  ; Robot abnormality
ANDNOT RB01_DSOUT9  ; Robot warning
AND 3811.08  ; ROBOT FAULT CLEAR TIMING
OUT 3811.09  ; COMPLETION OF ROBOT FAULT CLEAR
; rung 29
@LD RB01_DSOUT3  ; Robot abnormality
@OR RB01_DSOUT9  ; Robot warning
OR 3811.10  ; Robot abnormal code reading
ANDNOT RB01_DSOUT2  ; During robot operation
ANDNOT 3811.08  ; ROBOT FAULT CLEAR TIMING
ANDNOT 3811.12  ; Robot abnormal code reading reset
OUT 3811.10  ; Robot abnormal code reading
MOVD(083) #0 #210 3250  ; DATA AREA 1
MOV(021) #0 3251  ; DATA AREA 2
MOVD(083) #4 #0 3252  ; COMMAND AREA
TIM 0364 #2  ; Abnormal code reading timing
; rung 30
LD 3811.10  ; Robot abnormal code reading
AND T0364  ; Abnormal code reading timing
MOV(021) 3351 D520  ; Abnormal code storage area
; rung 31
LDNOT RB01_DSOUT3  ; Robot abnormality
ANDNOT RB01_DSOUT9  ; Robot warning
MOV(021) #0 D520  ; Abnormal code storage area

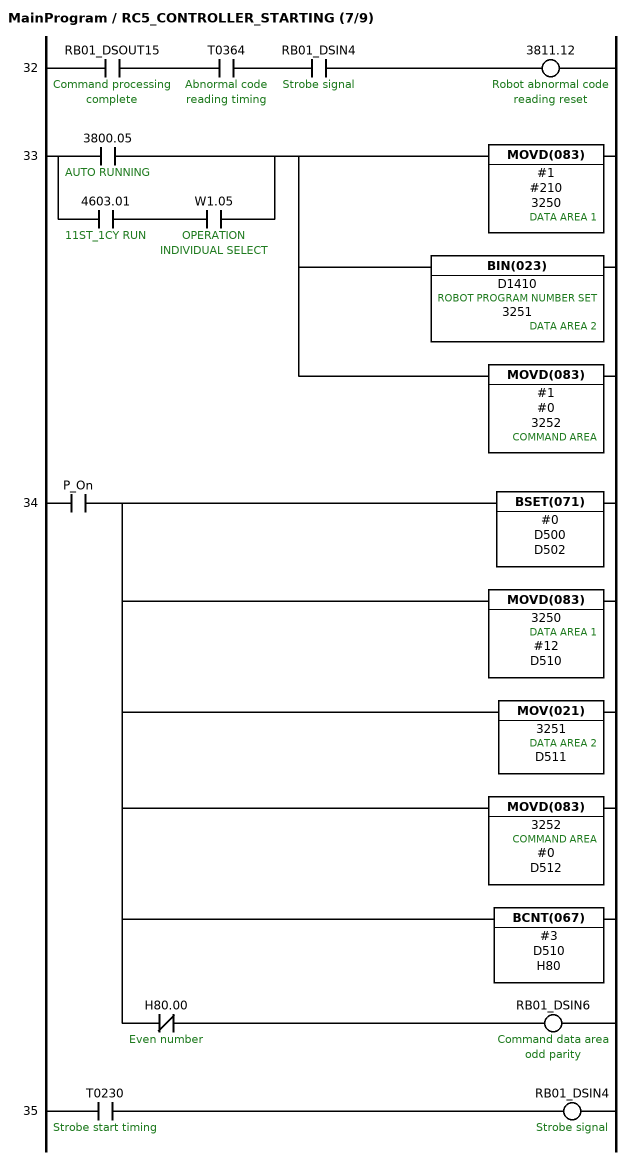
; rung 32
LD RB01_DSOUT15  ; Command processing complete
AND T0364  ; Abnormal code reading timing
AND RB01_DSIN4  ; Strobe signal
OUT 3811.12  ; Robot abnormal code reading reset
; rung 33
LD 3800.05  ; AUTO RUNNING
LD 4603.01  ; 11ST_1CY RUN
AND W1.05  ; OPERATION INDIVIDUAL SELECT
ORLD
MOVD(083) #1 #210 3250  ; DATA AREA 1
BIN(023) D1410 3251  ; ROBOT PROGRAM NUMBER SET, DATA AREA 2
MOVD(083) #1 #0 3252  ; COMMAND AREA
; rung 34
LD P_On
BSET(071) #0 D500 D502
MOVD(083) 3250 #12 D510  ; DATA AREA 1
MOV(021) 3251 D511  ; DATA AREA 2
MOVD(083) 3252 #0 D512  ; COMMAND AREA
BCNT(067) #3 D510 H80
ANDNOT H80.00  ; Even number
OUT RB01_DSIN6  ; Command data area odd parity
; rung 35
LD T0230  ; Strobe start timing
OUT RB01_DSIN4  ; Strobe signal

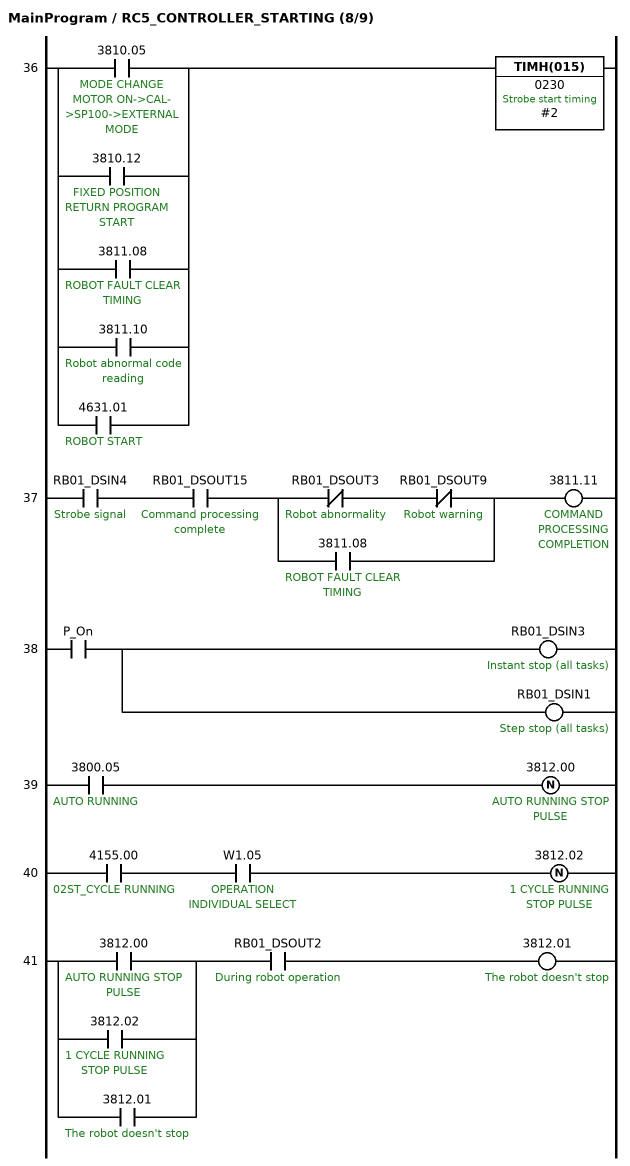
; rung 36
LD 3810.05  ; MODE CHANGE MOTOR ON->CAL->SP100->EXTERNAL MODE
OR 3810.12  ; FIXED POSITION RETURN PROGRAM START
OR 3811.08  ; ROBOT FAULT CLEAR TIMING
OR 3811.10  ; Robot abnormal code reading
OR 4631.01  ; ROBOT START
TIMH(015) 0230 #2  ; Strobe start timing
; rung 37
LD RB01_DSIN4  ; Strobe signal
AND RB01_DSOUT15  ; Command processing complete
LDNOT RB01_DSOUT3  ; Robot abnormality
ANDNOT RB01_DSOUT9  ; Robot warning
OR 3811.08  ; ROBOT FAULT CLEAR TIMING
ANDLD
OUT 3811.11  ; COMMAND PROCESSING COMPLETION
; rung 38
LD P_On
OUT RB01_DSIN3  ; Instant stop (all tasks)
OUT RB01_DSIN1  ; Step stop (all tasks)
; rung 39
LD 3800.05  ; AUTO RUNNING
DIFD(014) 3812.00  ; AUTO RUNNING STOP PULSE
; rung 40
LD 4155.00  ; 02ST_CYCLE RUNNING
AND W1.05  ; OPERATION INDIVIDUAL SELECT
DIFD(014) 3812.02  ; 1 CYCLE RUNNING STOP PULSE
; rung 41
LD 3812.00  ; AUTO RUNNING STOP PULSE
OR 3812.02  ; 1 CYCLE RUNNING STOP PULSE
OR 3812.01  ; The robot doesn't stop
AND RB01_DSOUT2  ; During robot operation
OUT 3812.01  ; The robot doesn't stop

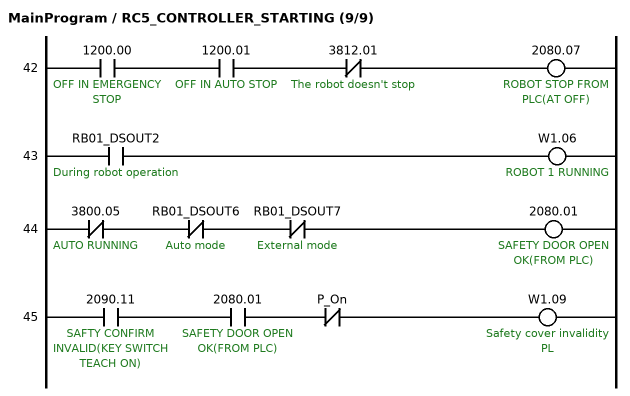
; rung 42
LD 1200.00  ; OFF IN EMERGENCY STOP
AND 1200.01  ; OFF IN AUTO STOP
ANDNOT 3812.01  ; The robot doesn't stop
OUT 2080.07  ; ROBOT STOP FROM PLC(AT OFF)
; rung 43
LD RB01_DSOUT2  ; During robot operation
OUT W1.06  ; ROBOT 1 RUNNING
; rung 44
LDNOT 3800.05  ; AUTO RUNNING
ANDNOT RB01_DSOUT6  ; Auto mode
ANDNOT RB01_DSOUT7  ; External mode
OUT 2080.01  ; SAFETY DOOR OPEN OK(FROM PLC)
; rung 45
LD 2090.11  ; SAFTY CONFIRM INVALID(KEY SWITCH TEACH ON)
AND 2080.01  ; SAFETY DOOR OPEN OK(FROM PLC)
ANDNOT P_On
OUT W1.09  ; Safety cover invalidity PL

### Section Servo_Motor

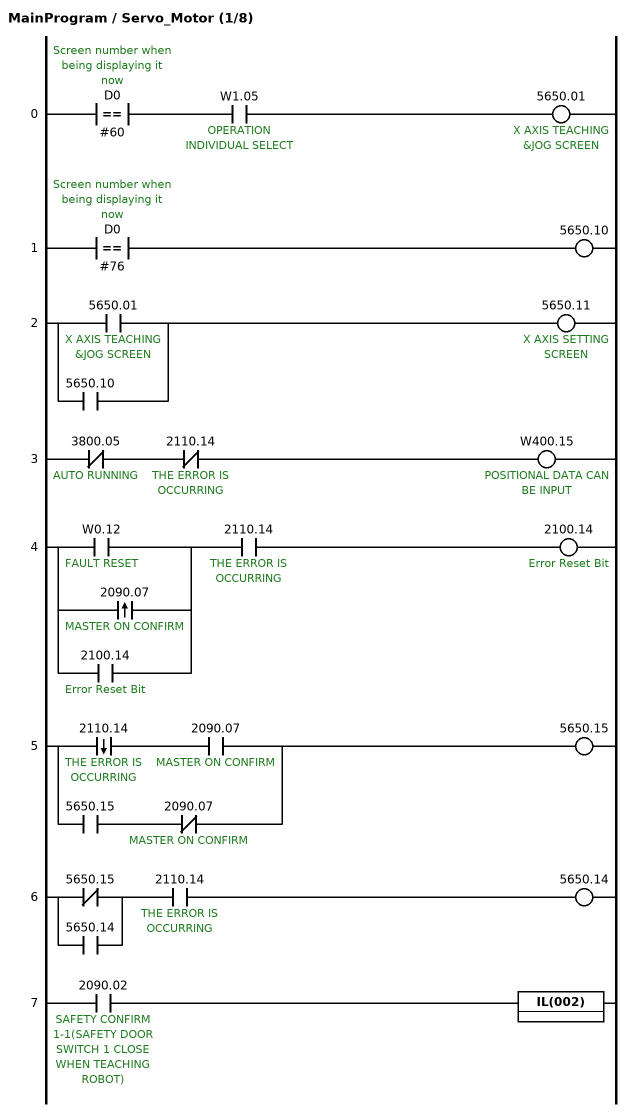
; rung 0
LD=(300) D0 #60  ; Screen number when being displaying it now
AND W1.05  ; OPERATION INDIVIDUAL SELECT
OUT 5650.01  ; X AXIS TEACHING &JOG SCREEN
; rung 1
LD=(300) D0 #76  ; Screen number when being displaying it now
OUT 5650.10
; rung 2
LD 5650.01  ; X AXIS TEACHING &JOG SCREEN
OR 5650.10
OUT 5650.11  ; X AXIS SETTING SCREEN
; rung 3
LDNOT 3800.05  ; AUTO RUNNING
ANDNOT 2110.14  ; THE ERROR IS OCCURRING
OUT W400.15  ; POSITIONAL DATA CAN BE INPUT
; rung 4
LD W0.12  ; FAULT RESET
@OR 2090.07  ; MASTER ON CONFIRM
OR 2100.14  ; Error Reset Bit
AND 2110.14  ; THE ERROR IS OCCURRING
OUT 2100.14  ; Error Reset Bit
; rung 5
%LD 2110.14  ; THE ERROR IS OCCURRING
AND 2090.07  ; MASTER ON CONFIRM
LD 5650.15
ANDNOT 2090.07  ; MASTER ON CONFIRM
ORLD
OUT 5650.15
; rung 6
LDNOT 5650.15
OR 5650.14
AND 2110.14  ; THE ERROR IS OCCURRING
OUT 5650.14
; rung 7
LD 2090.02  ; SAFETY CONFIRM 1-1(SAFETY DOOR SWITCH 1 CLOSE WHEN TEACHING ROBOT)
IL(002)

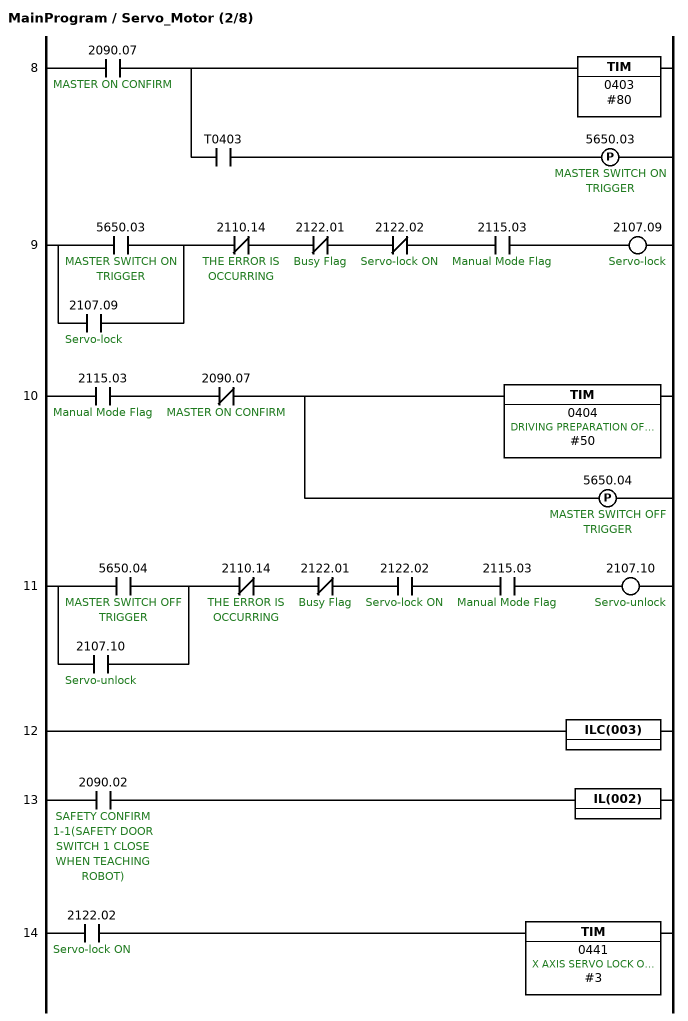
; rung 8
LD 2090.07  ; MASTER ON CONFIRM
TIM 0403 #80
AND T0403
DIFU(013) 5650.03  ; MASTER SWITCH ON TRIGGER
; rung 9
LD 5650.03  ; MASTER SWITCH ON TRIGGER
OR 2107.09  ; Servo-lock
ANDNOT 2110.14  ; THE ERROR IS OCCURRING
ANDNOT 2122.01  ; Busy Flag
ANDNOT 2122.02  ; Servo-lock ON
AND 2115.03  ; Manual Mode Flag
OUT 2107.09  ; Servo-lock
; rung 10
LD 2115.03  ; Manual Mode Flag
ANDNOT 2090.07  ; MASTER ON CONFIRM
TIM 0404 #50  ; DRIVING PREPARATION OFF CONFIRMATION
DIFU(013) 5650.04  ; MASTER SWITCH OFF TRIGGER
; rung 11
LD 5650.04  ; MASTER SWITCH OFF TRIGGER
OR 2107.10  ; Servo-unlock
ANDNOT 2110.14  ; THE ERROR IS OCCURRING
ANDNOT 2122.01  ; Busy Flag
AND 2122.02  ; Servo-lock ON
AND 2115.03  ; Manual Mode Flag
OUT 2107.10  ; Servo-unlock
; rung 12
ILC(003)
; rung 13
LD 2090.02  ; SAFETY CONFIRM 1-1(SAFETY DOOR SWITCH 1 CLOSE WHEN TEACHING ROBOT)
IL(002)
; rung 14
LD 2122.02  ; Servo-lock ON
TIM 0441 #3  ; X AXIS SERVO LOCK ON CONFIRMATION

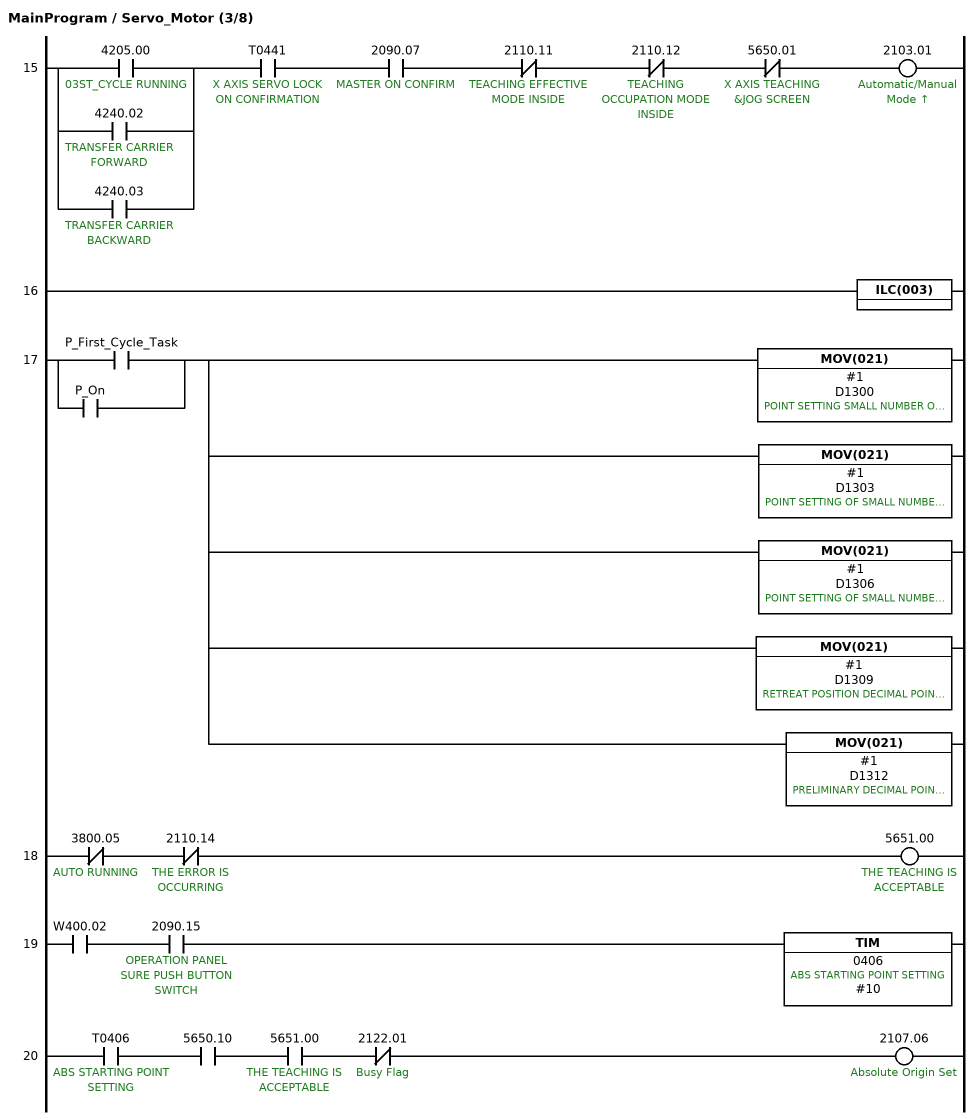
; rung 15
LD 4205.00  ; 03ST_CYCLE RUNNING
OR 4240.02  ; TRANSFER CARRIER FORWARD
OR 4240.03  ; TRANSFER CARRIER BACKWARD
AND T0441  ; X AXIS SERVO LOCK ON CONFIRMATION
AND 2090.07  ; MASTER ON CONFIRM
ANDNOT 2110.11  ; TEACHING EFFECTIVE MODE INSIDE
ANDNOT 2110.12  ; TEACHING OCCUPATION MODE INSIDE
ANDNOT 5650.01  ; X AXIS TEACHING &JOG SCREEN
OUT 2103.01  ; Automatic/Manual Mode ↑
; rung 16
ILC(003)
; rung 17
LD P_First_Cycle_Task
OR P_On
MOV(021) #1 D1300  ; POINT SETTING SMALL NUMBER OF FORWARD SPEEDS
MOV(021) #1 D1303  ; POINT SETTING OF SMALL NUMBER OF ADVANCEMENT EDGES
MOV(021) #1 D1306  ; POINT SETTING OF SMALL NUMBER OF RETREAT SPEEDS
MOV(021) #1 D1309  ; RETREAT POSITION DECIMAL POINT SETTING
MOV(021) #1 D1312  ; PRELIMINARY DECIMAL POINT SETTING
; rung 18
LDNOT 3800.05  ; AUTO RUNNING
ANDNOT 2110.14  ; THE ERROR IS OCCURRING
OUT 5651.00  ; THE TEACHING IS ACCEPTABLE
; rung 19
LD W400.02
AND 2090.15  ; OPERATION PANEL SURE PUSH BUTTON SWITCH
TIM 0406 #10  ; ABS STARTING POINT SETTING
; rung 20
LD T0406  ; ABS STARTING POINT SETTING
AND 5650.10
AND 5651.00  ; THE TEACHING IS ACCEPTABLE
ANDNOT 2122.01  ; Busy Flag
OUT 2107.06  ; Absolute Origin Set

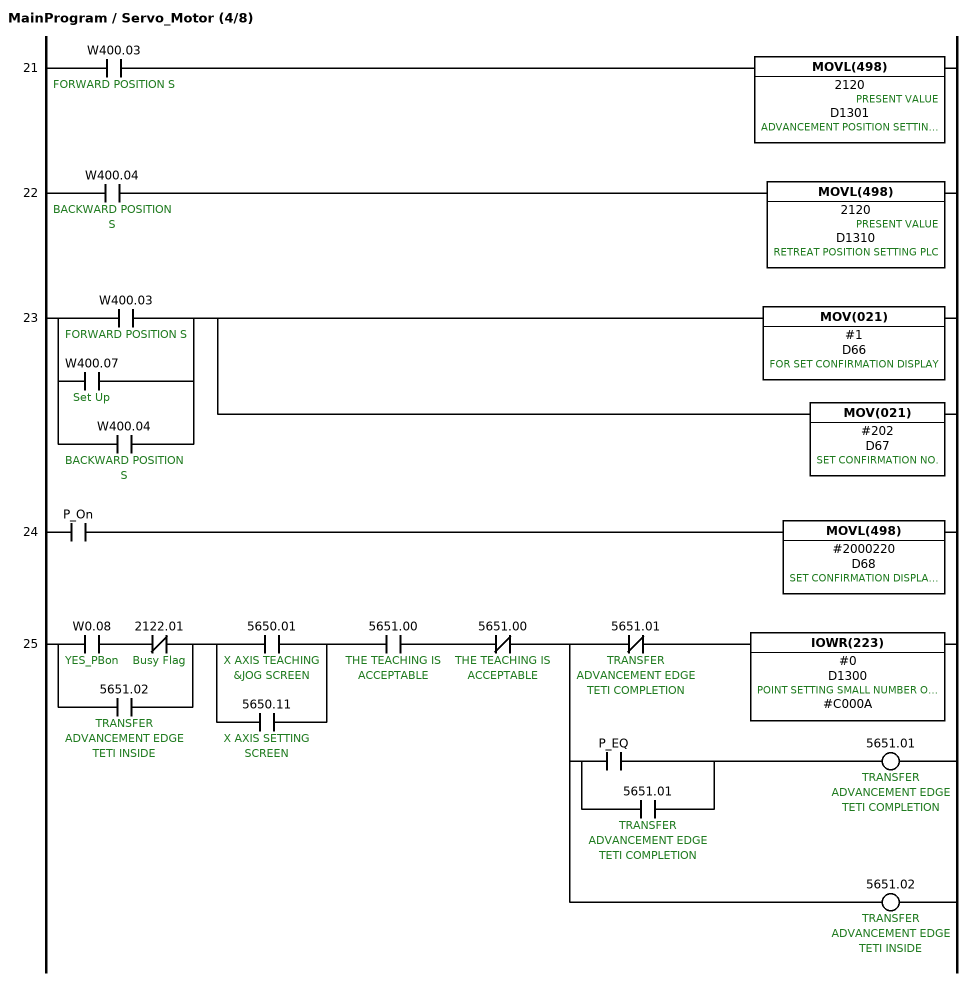
; rung 21
LD W400.03  ; FORWARD POSITION S
MOVL(498) 2120 D1301  ; PRESENT VALUE, ADVANCEMENT POSITION SETTING PLC
; rung 22
LD W400.04  ; BACKWARD POSITION S
MOVL(498) 2120 D1310  ; PRESENT VALUE, RETREAT POSITION SETTING PLC
; rung 23
LD W400.03  ; FORWARD POSITION S
OR W400.07  ; Set Up
OR W400.04  ; BACKWARD POSITION S
MOV(021) #1 D66  ; FOR SET CONFIRMATION DISPLAY
MOV(021) #202 D67  ; SET CONFIRMATION NO.
; rung 24
LD P_On
MOVL(498) #2000220 D68  ; SET CONFIRMATION DISPLAY POSITION
; rung 25
LD W0.08  ; YES_PBon
ANDNOT 2122.01  ; Busy Flag
OR 5651.02  ; TRANSFER ADVANCEMENT EDGE TETI INSIDE
LD 5650.01  ; X AXIS TEACHING &JOG SCREEN
OR 5650.11  ; X AXIS SETTING SCREEN
ANDLD
AND 5651.00  ; THE TEACHING IS ACCEPTABLE
ANDNOT 5651.00  ; THE TEACHING IS ACCEPTABLE
OUT TR0
ANDNOT 5651.01  ; TRANSFER ADVANCEMENT EDGE TETI COMPLETION
IOWR(223) #0 D1300 #C000A  ; POINT SETTING SMALL NUMBER OF FORWARD SPEEDS
LD TR0
LD P_EQ
OR 5651.01  ; TRANSFER ADVANCEMENT EDGE TETI COMPLETION
ANDLD
OUT 5651.01  ; TRANSFER ADVANCEMENT EDGE TETI COMPLETION
LD TR0
OUT 5651.02  ; TRANSFER ADVANCEMENT EDGE TETI INSIDE

